// TwinCAT 3 PLC project LightSample
// ProgramVersion: 3.1.4020.1
// libraries:
//   Tc2_Standard, * (Beckhoff Automation GmbH)
//   Tc2_System, * (Beckhoff Automation GmbH)
//   Tc3_Interfaces, * (Beckhoff Automation GmbH)
//   Tc3_Module, * (Beckhoff Automation GmbH)
// project tree:
//   / PlcTask.TcTTO
//   POUs/ FB_LightControl.TcPOU, FB_StairwellLight.TcPOU, FB_StandardLight.TcPOU, ILight.TcIO, MAIN.TcPOU
// real-time tasks:
//   TASK PlcTask: cycle T#10ms, priority 20, ADS port 350

CONFIGURATION LightSample
    RESOURCE PLC ON TwinCAT3
        TASK PlcTask(INTERVAL := T#10ms, PRIORITY := 20);
        PROGRAM MAIN WITH PlcTask : MAIN;
    END_RESOURCE
END_CONFIGURATION

// ---- POUs/ILight.TcIO
INTERFACE ILight

METHOD M_Off
END_METHOD

PROPERTY P_ControlValue : BOOL
SET
END_SET
GET
END_GET
END_PROPERTY

METHOD M_On
END_METHOD

METHOD M_Execution
END_METHOD

END_INTERFACE

// ---- POUs/MAIN.TcPOU
PROGRAM MAIN
VAR
	fbLightControlRoom01	: FB_LightControl;
	bSwitchOn01				: BOOL;
	bSwitchOff01			: BOOL;
	bValue01				: BOOL;
	fbStandardLight			: FB_StandardLight;
	fbLightControlRoom02	: FB_LightControl;
	bSwitchOn02				: BOOL;
	bSwitchOff02			: BOOL;
	bValue02				: BOOL;
	fbStairwellLight		: FB_StairwellLight;
END_VAR

fbLightControlRoom01(bOn := bSwitchOn01, 
					 bOff := bSwitchOff01, 
					 LightType := fbStandardLight,
					 bControlValue => bValue01);

fbLightControlRoom02(bOn := bSwitchOn02, 
					 bOff := bSwitchOff02, 
					 LightType := fbStairwellLight,
					 bControlValue => bValue02);

END_PROGRAM

// ---- POUs/FB_LightControl.TcPOU
FUNCTION_BLOCK FB_LightControl
VAR_INPUT
	bOn				: BOOL;
	bOff			: BOOL;
	LightType		: ILight;
END_VAR
VAR_OUTPUT
	bControlValue	: BOOL;
END_VAR
VAR
	rtrigOn			: R_TRIG;
	rtrigOff		: R_TRIG;
END_VAR

rtrigOn(CLK := bOn);
rtrigOff(CLK := bOff);

IF (rtrigOn.Q) THEN
	LightType.M_On();
END_IF

IF (rtrigOff.Q) THEN
	LightType.M_Off();
END_IF

LightType.M_Execution();
bControlValue := LightType.P_ControlValue;

END_FUNCTION_BLOCK

// ---- POUs/FB_StandardLight.TcPOU
FUNCTION_BLOCK FB_StandardLight IMPLEMENTS ILight
VAR
	bControlValue	: BOOL;
END_VAR

METHOD M_On
P_ControlValue := TRUE;
END_METHOD

METHOD M_Off
P_ControlValue := FALSE;
END_METHOD

PROPERTY P_ControlValue : BOOL
GET
P_ControlValue := bControlValue;
END_GET
SET
bControlValue := P_ControlValue;
END_SET
END_PROPERTY

METHOD M_Execution
END_METHOD

END_FUNCTION_BLOCK

// ---- POUs/FB_StairwellLight.TcPOU
FUNCTION_BLOCK FB_StairwellLight IMPLEMENTS ILight
VAR
	bControlValue		: BOOL;
	fbTon				: TON := (PT := TIME#3s0ms);
END_VAR

METHOD M_Execution
fbTon();
IF (fbTon.Q) THEN
	THIS^.M_Off();
END_IF
END_METHOD

PROPERTY P_ControlValue : BOOL
GET
P_ControlValue := bControlValue;
END_GET
SET
bControlValue := P_ControlValue;
END_SET
END_PROPERTY

METHOD M_On
P_ControlValue := TRUE;
fbTon(IN := TRUE);
END_METHOD

METHOD M_Off
P_ControlValue := FALSE;
fbTon(IN := FALSE);
END_METHOD

END_FUNCTION_BLOCK
